FUNCTION F_ITC_SendGCR : BOOL
(**************************************************************************************
 * 	Application		:	BoxControl Framework
 *	Revision		:	$Revision: 404529 $
 *	Revision date	:	$Date: 2018-04-23 08:21:38 +0200 (Mo., 23 Apr 2018) $
 *	Last changed by	:	$Author: b7bolm $
 *	URL				:	$URL: http://almscdc.swisslog.com/repo/SWPD/Development/BoxControlFramework/20_Release/trunk/01_Software/BCF/BCF/JumpStart/20_Product/10_App/11_Com/10_Lib/10_Conv/11_ITC/F_ITC_SendGCR.TcPOU $
 *
 *	Purpose			:	Wrap message - GCR
 *
 * ------------------------------------------------------------------------------------
 *	Copyright Swisslog [IP AG], Switzerland. All rights reserved.
 * 
 * ------------------------------------------------------------------------------------
 *	
 * 	Revision History: 
 *
 * 	VERSION			DATE			INITIALS			DESCRIPTION
 *	0.1				01.01.2001		swl					Example
 *
 **************************************************************************************)
VAR_INPUT
	eChannelSrc		: E_MFCS_Channel; // Source communicaton channel	
	GroupName		: STRING(Conveyor.POSITION_STRINGLENGTH); // SIS Group Name MM-GGG-0000-000
	Code			: INT; // Control code
	Variable		: DINT; // Control code variable
	eReturnCode		: E_ErrorConv; // Return code
END_VAR
VAR
	GCR				: ST_ITC_GCR; 
END_VAR

// Map values
GCR.GroupName := GroupName;
GCR.Code := Code;
GCR.Variable := Variable;
GCR.ReturnCode := eReturnCode;

// Forward to ITC
F_ITC_SendGCR := fbITC_Manager.M_SendData(
					meChannel	:= eChannelSrc,
					mMsgType	:= E_ITC_MsgTypeConv.GROUP_CONTROL_REPLY,
					mpData		:= ADR(GCR),
					mLen		:= SIZEOF(GCR));

END_FUNCTION

(* stored: Version 1.1.0.1, ProductVersion 3.1.4022.12
   POU F_ITC_SendGCR: Id {d5218ab7-de9c-45ce-89ef-ee513a952058}, SpecialFunc None *)
